{attribute 'qualified_only'}
{attribute 'strict'}
{attribute 'to_string'}
TYPE LogLevel :
(
	Debug := 0,
	Information := 1,
	Warning := 2,
	Error := 3,
	Fatal := 4
);
END_TYPE

(* stored: Version 1.1.0.1
   DUT LogLevel: Id {55156f2d-d00f-48d6-bde4-ddbebdef9a67} *)
